(* IEC 61131-3 sources: eCockpitGit/test_project/src/%F%00 Library/%F%Structured Buffer Read Write Base/%ITF%ITF_StructReaderBase/%F%Reading, 3 files *)

(* ---- %METH%compareString.st ---- *)
//This method compares a string to the selected string
METHOD compareString : BOOL
VAR_INPUT
	str				:POINTER TO EASCII;
END_VAR
(*%!%__DELIMITER__%!%*)

(* ---- %METH%exportValue.st ---- *)
//This method returns the buffer position and size of the currently selected struct/object
METHOD exportValue : BOOL
VAR_OUTPUT
	position		:POINTER TO EASCII;
	size			:DWORD;
END_VAR
(*%!%__DELIMITER__%!%*)

(* ---- %METH%readString.st ---- *)
//This method returns the string value of the currently selected item
//Returns true on output if value is valid
METHOD readString
VAR_INPUT
	str		:POINTER TO EASCII;		//Address of the name to find, only input string address or zero terminated byte array
	lenMax	:DWORD;					//Max lenght of string value
END_VAR
VAR_OUTPUT
	len		:WORD;					//Actual lenght of string value
END_VAR
(*%!%__DELIMITER__%!%*)
